Staubli VAL3: onF7Event.pgx

program onF7Event()
  local num local1
  local string l_sPage
  local string l_sItem
begin
  // look if the bButton is enable
  if bButton[6]
    //
    if saveData:mode==0
      call passwd()
      call use:nullKey(nKey)
    else
      l_sPage="Disk://kernel/page/advance"
      call loadPage(l_sPage,l_sItem)
      logMsg("[KERNEL] INTERFACE:PAGE Home Page")
    endIf
  endIf
end
